FUNCTION_BLOCK 
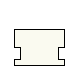
  VAR
     : ;
     : ;
     : ;
  END_VAR
  ALGORITHM ALG IN ST:

  END_ALGORITHM
END_FUNCTION_BLOCK
(* other elements stored in the file *)
(* ECState name=START Initial=true *)
(* ECState name=BODY *)
(* ECAction Algorithm=ALG *)
